// TIA Portal V19 program export: 1 tag tables, 1 data types, 2 data blocks, 10 code blocks (in call order from the OBs), 4 instance data blocks

VAR_GLOBAL   // PLC tag table "DefaultTagTable"
   Tag_1 AT %M20.7 : Bool;
END_VAR

TYPE "typeStartLift"
TITLE = typeStartLift
// PLC data type start lift
   STRUCT
      startLiftUp : Bool;   // Start lift up
      startLiftDown : Bool;   // Start lift down
   END_STRUCT;
END_TYPE

DATA_BLOCK "Actions"   // DB3
{ S7_Optimized_Access := 'TRUE' }
// stored: MemoryReserve 100
   VAR
      Action_AirComprID1 : String := 'Check that no emergency stop has been depressed. If it has, check why. The machine is now ready to start with the Unit On button. The alarm is reset automatically when the cause is removed (logically controlled).';
      TextList : DWord;
      Trigger : UInt;
      Ack : Bool;
   END_VAR
BEGIN
END_DATA_BLOCK

DATA_BLOCK "SeqData"   // DB11
TITLE = SeqData
{ S7_Optimized_Access := 'TRUE'; DB_Accessible_From_OPC_UA := 'FALSE' }
AUTHOR : Siemens
// Global DB for BeltLift
// stored: DBAccessibleFromOPCUA false, MemoryReserve 100
   VAR
      plantOn : Bool := true;   // Plant switched on
      compressedAir : Bool;   // Druckluft nicht in Ordnung. Im Fehlerfall ist die Ursache: Der zur Maschine gehörende Not-Halt hat die Maschine gestoppt. Bei ausgeschalteter Maschine oder gedrücktem Not-Halt können keine Funktionen ausgeführt werden. / Compressed air not OK. In case of an Error Cause: The emergency stop belonging to the machine has stopped the machine. No functions can be performed when the machine is shut off or the emergency stop is pressed.
      powerVoltage : Bool;   // Spannungsversorgung nicht in Ordnung. Im Fehlerfall ist die Druckluft nicht in Ordnung. Im Fehlerfall ist die Ursache: Der zur Maschine gehörende Not-Halt hat die Maschine gestoppt. Bei ausgeschalteter Maschine oder gedrücktem Not-Halt können keine Funktionen ausgeführt werden. / Voltage power supply not OK.
      doorClosed : Bool;   // Safety door closed
      autoStart : Bool;   // Automatic start
      autoStop : Bool;   // Automatic stop
      autoStarted : Bool := false;   // Automatic started
      autoStopped : Bool;   // Automatic stopped
      ackSeq : Bool;   // Acknowledge GRAPH FB
      errFltSeq : Bool;   // Error Graph FB
      seqStart : Bool;   // GRAPH sequence started
      newCase : Bool;   // Sensor new case
      posCaseBelt : Int;   // Case position on belt
      posLift1 : Int;   // Lift 1 position
      posLift2 : Int;   // Lift 2 position
      visCaseLift1 : Bool;   // Case lift1 visible
      visCaseLift2 : Bool;   // Case lift2 visible
      setStop1 : Bool;   // Set stopper1
      setStop2 : Bool;   // Set stopper2
      sensorStop1 : Bool;   // Sensor at stopper1
      sensorStop2 : Bool;   // Sensor at stopper2
      sensorStop3 : Bool;   // Sensor at stopper3
      errSensorStop1 : Bool;   // Error on Sensor at stopper1
      errSensorStop2 : Bool;   // Error on Sensor at stopper2
      errSensorStop3 : Bool;   // Error on Sensor at stopper2
      errSensorNewCase : Bool;   // Error on Sensor at new case
      toLift1 : Bool;   // Case to lift1 or lift2
      autoLift1 : "typeStartLift";   // Start automatic lift1
      autoLift2 : "typeStartLift";   // Start automatic lift2
      manLift1 : "typeStartLift";   // Start manual lift1
      manLift2 : "typeStartLift";   // Start manual lift2
      outLift1Up : Bool;   // Output lift1 up
      outLift1Down : Bool;   // Output lift1 down
      outLift2Up : Bool;   // Output lift2 up
      outLift2Down : Bool;   // Output lift2 down
      sensorLift1Up : Bool;   // Sensor lift1 up
      sensorLift1Down : Bool;   // Sensor lift1 down
      sensorLift2Up : Bool;   // Sensor lift2 up
      sensorLift2Down : Bool;   // Sensor lift2 down
      simOperandSupVis : Bool;   // Simulation supervision operand
      simInterlockSupVis : Bool;   // Simulation supervision interlock
      simLiftFreeSupVis : Bool;   // Simulation supervision lift free
      simActReactSupVis : Bool;   // Simulation supervision action and reaction
      simPositionSupVis : Bool;   // Simulation supervision position
      simUdtOperandSupVis : Bool;   // Simulation supervision operand in UDT
      simActive : Bool;   // Simulation active
      releaseSimPlantOn : Bool;   // Release simulation plant on
      releaseSimAutoStarted : Bool;   // Release simulation auto started
      releaseSimAutoStopped : Bool;   // Release simulation auto stopped
      beltLEDs : Word;   // Moving lights belt
      lift1LEDs : Word;   // Moving lights lift1
      lift2LEDs : Word;   // Moving lights lift2
      stateCase : Array[0..3] of Bool;   // State case position
      liftFree : Bool := true;   // Lift is free for new case / Lift ist bereit für einen neuen Kasten
      simInterlockSupVisLiftFree : Bool;   // Simulation supervision interlock / Simulation supervision interlock lift free
      resetCrit : Bool;
      identTimeStamp : LDT;
      retVal : Int;
      frequency : Real := 10.0;
      freqError : Bool;
      freqStatus : Word;
      textListID { ExternalAccessible := 'False'; ExternalVisible := 'False'; ExternalWritable := 'False'} : Word;
   END_VAR
BEGIN
END_DATA_BLOCK

ORGANIZATION_BLOCK "Main"   // OB1, LAD, ProgramCycle
TITLE = "Main Program Sweep (Cycle)"
{ S7_Optimized_Access := 'TRUE' }
AUTHOR : Siemens
// "Main Program
// stored: IsIECCheckEnabled true, SetENOAutomatically true
   VAR_INPUT
      Initial_Call : Bool;   // Initial call of this OB
      Remanence : Bool;   // =True, if remanent data are available
   END_VAR
BEGIN

REGION Network 1
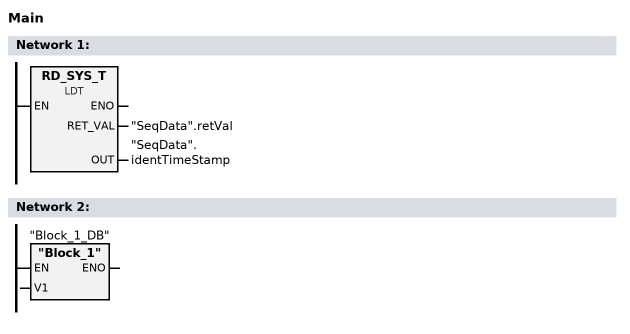
   RUNG wire#powerrail
      { S7_Templates := "date_type := LDT" } RD_SYS_T(RET_VAL => "SeqData".retVal, OUT => "SeqData".identTimeStamp)
   END_RUNG
   // the same network as SCL:
   "SeqData".retVal := RD_SYS_T(OUT => "SeqData".identTimeStamp);
END_REGION

REGION Network 2
   RUNG wire#powerrail
      "Block_1_DB"(V1 :=)
   END_RUNG
   // the same network as SCL:
   "Block_1_DB"();   // "Block_1"
END_REGION
END_ORGANIZATION_BLOCK

ORGANIZATION_BLOCK "MainBeltLift"   // OB125, FBD, ProgramCycle
TITLE = "Main Program Sweep (Cycle)"
{ S7_Optimized_Access := 'TRUE' }
AUTHOR : Siemens
// Main programm belt lift
// stored: IsIECCheckEnabled true, SetENOAutomatically true
   VAR_INPUT
      Initial_Call : Bool;   // Initial call of this OB
      Remanence : Bool;   // =True, if remanent data are available
   END_VAR
BEGIN

REGION Network 1
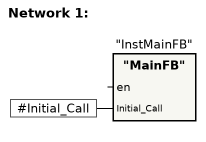
   "InstMainFB"(Initial_Call := #Initial_Call);   // "MainFB"
END_REGION
END_ORGANIZATION_BLOCK

FUNCTION_BLOCK "MainFB"   // FB10, FBD
TITLE = MainFB
{ S7_Optimized_Access := 'TRUE' }
AUTHOR : Siemens
// Main FB BeltLift
// stored: IsIECCheckEnabled true, MemoryReserve 100, SetENOAutomatically true
   VAR_INPUT
      Initial_Call { ExternalAccessible := 'False'; ExternalVisible := 'False'; ExternalWritable := 'False'} : Bool;   // Initial call of this OB
   END_VAR
   VAR
      instCommon { ExternalAccessible := 'False'; ExternalVisible := 'False'; ExternalWritable := 'False'; S7_SetPoint := 'True'} : "Common";
      instLift1Cmd { ExternalAccessible := 'False'; ExternalVisible := 'False'; ExternalWritable := 'False'; S7_SetPoint := 'True'} : "LiftCmd";
      instLift2Cmd { ExternalAccessible := 'False'; ExternalVisible := 'False'; ExternalWritable := 'False'; S7_SetPoint := 'True'} : "LiftCmd";
      instLiftSim { ExternalAccessible := 'False'; ExternalVisible := 'False'; ExternalWritable := 'False'; S7_SetPoint := 'True'} : "LiftSim";
   END_VAR
BEGIN

REGION Network 1: common
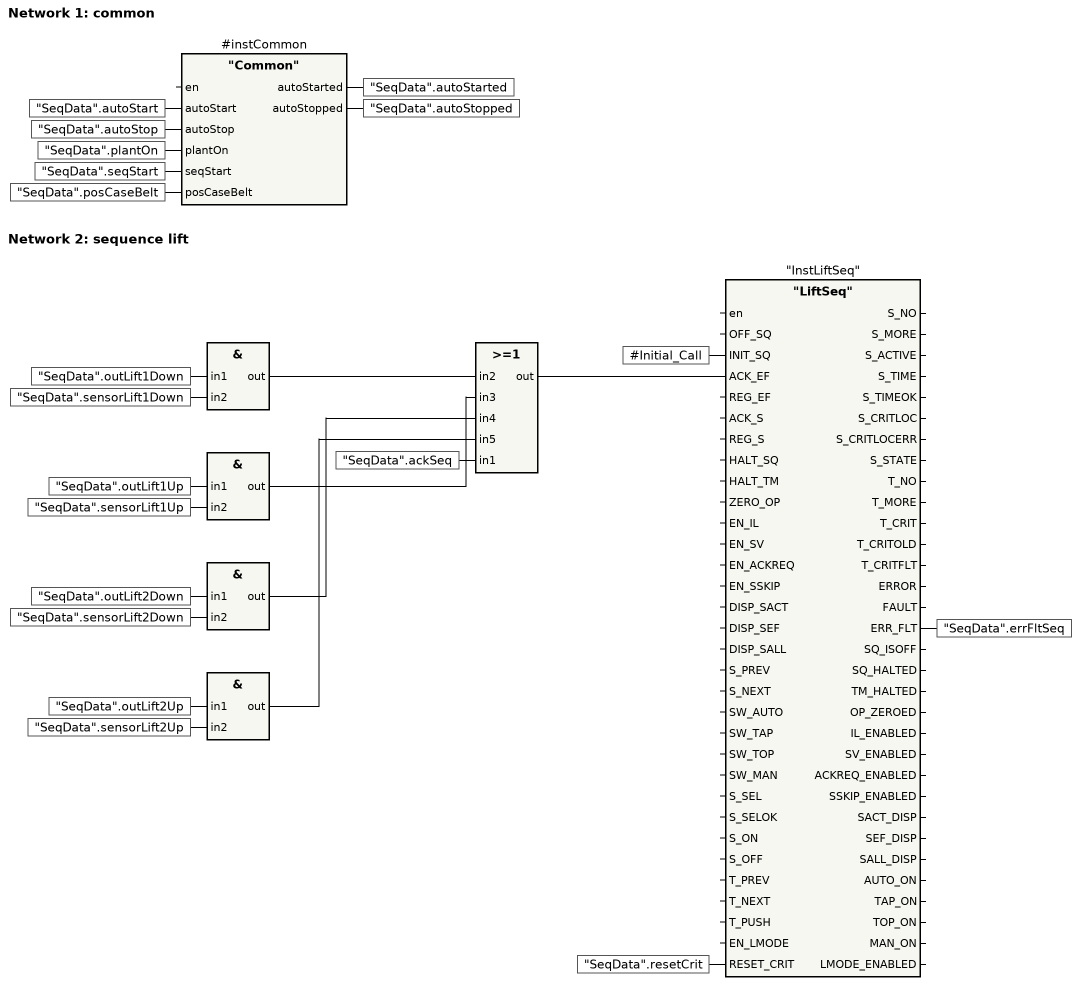
   #instCommon(autoStart := "SeqData".autoStart,   // "Common"
               autoStop := "SeqData".autoStop,
               plantOn := "SeqData".plantOn,
               seqStart := "SeqData".seqStart,
               posCaseBelt := "SeqData".posCaseBelt,
               autoStarted => "SeqData".autoStarted,
               autoStopped => "SeqData".autoStopped);
END_REGION

REGION Network 2: sequence lift
   "InstLiftSeq"(INIT_SQ := #Initial_Call,   // "LiftSeq"
                 ACK_EF := ("SeqData".outLift1Down AND "SeqData".sensorLift1Down) OR ("SeqData".outLift1Up AND "SeqData".sensorLift1Up) OR ("SeqData".outLift2Down AND "SeqData".sensorLift2Down) OR ("SeqData".outLift2Up AND "SeqData".sensorLift2Up) OR "SeqData".ackSeq,
                 RESET_CRIT := "SeqData".resetCrit,
                 ERR_FLT => "SeqData".errFltSeq);
END_REGION

REGION Network 3: Lift 1
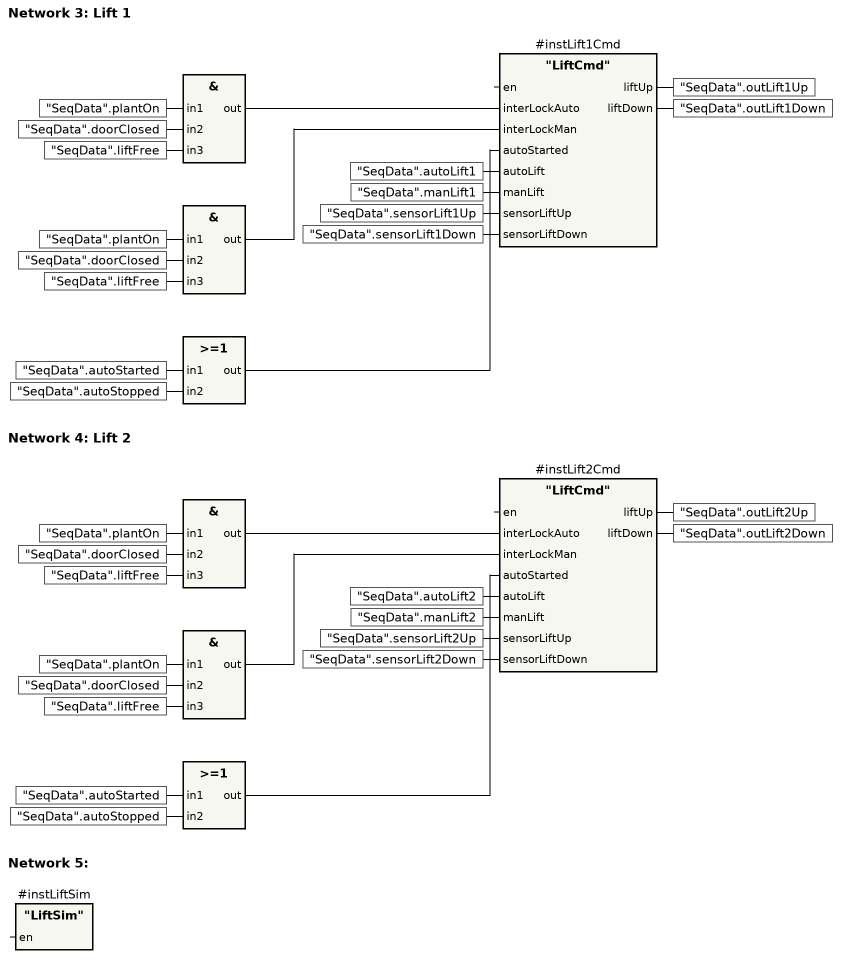
   #instLift1Cmd(interLockAuto := "SeqData".plantOn AND "SeqData".doorClosed AND "SeqData".liftFree,   // "LiftCmd"
                 interLockMan := "SeqData".plantOn AND "SeqData".doorClosed AND "SeqData".liftFree,
                 autoStarted := "SeqData".autoStarted OR "SeqData".autoStopped,
                 autoLift := "SeqData".autoLift1,
                 manLift := "SeqData".manLift1,
                 sensorLiftUp := "SeqData".sensorLift1Up,
                 sensorLiftDown := "SeqData".sensorLift1Down,
                 liftUp => "SeqData".outLift1Up,
                 liftDown => "SeqData".outLift1Down);
END_REGION

REGION Network 4: Lift 2
   #instLift2Cmd(interLockAuto := "SeqData".plantOn AND "SeqData".doorClosed AND "SeqData".liftFree,   // "LiftCmd"
                 interLockMan := "SeqData".plantOn AND "SeqData".doorClosed AND "SeqData".liftFree,
                 autoStarted := "SeqData".autoStarted OR "SeqData".autoStopped,
                 autoLift := "SeqData".autoLift2,
                 manLift := "SeqData".manLift2,
                 sensorLiftUp := "SeqData".sensorLift2Up,
                 sensorLiftDown := "SeqData".sensorLift2Down,
                 liftUp => "SeqData".outLift2Up,
                 liftDown => "SeqData".outLift2Down);
END_REGION

REGION Network 5
   #instLiftSim();   // "LiftSim"
END_REGION
END_FUNCTION_BLOCK

FUNCTION_BLOCK "Common"   // FB13, FBD
TITLE = Common
{ S7_Optimized_Access := 'TRUE' }
AUTHOR : Siemens
// Common functions BeltLift
// stored: IsIECCheckEnabled true, MemoryReserve 100, SetENOAutomatically true
   VAR_INPUT
      autoStart { ExternalAccessible := 'False'; ExternalVisible := 'False'; ExternalWritable := 'False'} : Bool;
      autoStop { ExternalAccessible := 'False'; ExternalVisible := 'False'; ExternalWritable := 'False'} : Bool;
      plantOn { ExternalAccessible := 'False'; ExternalVisible := 'False'; ExternalWritable := 'False'} : Bool;
      seqStart { ExternalAccessible := 'False'; ExternalVisible := 'False'; ExternalWritable := 'False'} : Bool;
      posCaseBelt { ExternalAccessible := 'False'; ExternalVisible := 'False'; ExternalWritable := 'False'} : Int;
   END_VAR
   VAR_OUTPUT
      autoStarted { ExternalAccessible := 'False'; ExternalVisible := 'False'; ExternalWritable := 'False'} : Bool;
      autoStopped { ExternalAccessible := 'False'; ExternalVisible := 'False'; ExternalWritable := 'False'} : Bool;
   END_VAR
   VAR
      statCaseOnStopper { ExternalAccessible := 'False'; ExternalVisible := 'False'; ExternalWritable := 'False'} : Bool;
      statAutoStopped { ExternalAccessible := 'False'; ExternalVisible := 'False'; ExternalWritable := 'False'} : Bool;
   END_VAR
BEGIN

REGION Network 1
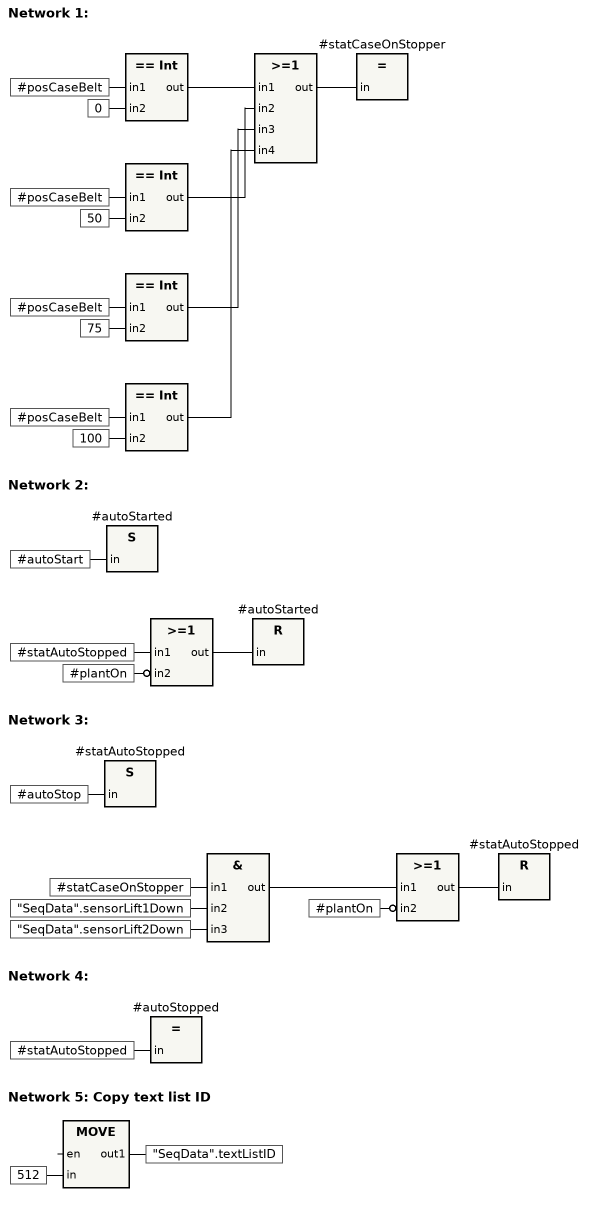
   #statCaseOnStopper := (#posCaseBelt = 0) OR (#posCaseBelt = 50) OR (#posCaseBelt = 75) OR (#posCaseBelt = 100);
END_REGION

REGION Network 2
   IF #autoStart THEN #autoStarted := TRUE; END_IF;
   IF #statAutoStopped OR NOT #plantOn THEN #autoStarted := FALSE; END_IF;
END_REGION

REGION Network 3
   IF #autoStop THEN #statAutoStopped := TRUE; END_IF;
   IF (#statCaseOnStopper AND "SeqData".sensorLift1Down AND "SeqData".sensorLift2Down) OR NOT #plantOn THEN
       #statAutoStopped := FALSE;
   END_IF;
END_REGION

REGION Network 4
   #autoStopped := #statAutoStopped;
END_REGION

REGION Network 5: Copy text list ID
   "SeqData".textListID := 512;
END_REGION
END_FUNCTION_BLOCK

FUNCTION_BLOCK "LiftSeq"   // FB12, GRAPH
TITLE = LiftSeq
AUTHOR : Siemens
// Graph sequence BeltLift
// stored: GraphVersion 6.0, InitialValuesAcquisition true, IsIECCheckEnabled true, LanguageInNetworks FBD, SetENOAutomatically true
   // inherited from GRAPH_BASE
   VAR_INPUT
      OFF_SQ { ExternalWritable := 'False'} : Bool := false;   // Kette ausschalten / Turn sequence off
      INIT_SQ { ExternalWritable := 'False'} : Bool := false;   // Kette in Initialzustand versetzen / Set sequence to initial state
      ACK_EF { ExternalWritable := 'False'} : Bool := false;   // Alle Fehler und Störungen quittieren / Acknowledge all errors and faults
      REG_EF { ExternalWritable := 'False'} : Bool := false;   // Register all errors and faults / Alle Fehler und Störungen registrieren
      ACK_S { ExternalWritable := 'False'} : Bool := false;   // Acknowledge step indicated in S_NO / Schritt quittieren, der an Parameter S_NO anliegt
      REG_S { ExternalWritable := 'False'} : Bool := false;   // Register the step indicated in S_NO / Schritt registrieren, der an Parameter S_NO anliegt
      HALT_SQ { ExternalWritable := 'False'} : Bool := false;   // Halt sequence immediately / Kette sofort anhalten
      HALT_TM { ExternalWritable := 'False'} : Bool := false;   // Halt timers immediately / Zeiten sofort anhalten
      ZERO_OP { ExternalWritable := 'False'} : Bool := false;   // Set all operands assigned with N, L, D to 0 / Alle mit N, L, D zugewiesenen Operanden auf 0 setzen
      EN_IL { ExternalWritable := 'False'} : Bool := false;   // Activate interlocks / Interlockbearbeitung aktivieren
      EN_SV { ExternalWritable := 'False'} : Bool := false;   // Activate supervision processing / Supervisionsbearbeitung aktivieren
      EN_ACKREQ { ExternalWritable := 'False'} : Bool := false;   // Activate mandatory acknowledgment / Quittierpflicht aktivieren
      EN_SSKIP { ExternalWritable := 'False'} : Bool := false;   // Enable "Skip step" / "Schritte überspringen" aktivieren
      DISP_SACT { ExternalWritable := 'False'} : Bool := false;   // Display active steps only / Nur aktive Schritte anzeigen
      DISP_SEF { ExternalWritable := 'False'} : Bool := false;   // Display only steps with errors and disrupted steps / Nur fehlerhafte und gestörte Schritte anzeigen
      DISP_SALL { ExternalWritable := 'False'} : Bool := false;   // Display all steps / Alle Schritte anzeigen
      S_PREV { ExternalWritable := 'False'} : Bool := false;   // Vorherigen Schritt am Parameter S_NO ausgeben / Output previous step in parameter S_NO
      S_NEXT { ExternalWritable := 'False'} : Bool := false;   // Nächsten Schritt am Parameter S_NO anzeigen / Indicate next step in parameter S_NO
      SW_AUTO { ExternalWritable := 'False'} : Bool := false;   // Automtischer Betrieb / Automatic mode
      SW_TAP { ExternalWritable := 'False'} : Bool := false;   // Halbautomatisch/Weiterschalten mit Transition / Semiautomatic/switch with transition
      SW_TOP { ExternalWritable := 'False'} : Bool := false;   // Halbautomatisch/Ignoriere Transition / Semiautomatic/ignore transition
      SW_MAN { ExternalWritable := 'False'} : Bool := false;   // Handbetrieb / Manual mode
      S_SEL { ExternalWritable := 'False'} : Int := 0;   // Schritt auswählen, der an S_NO ausgegeben werden soll / Select step to be output to S_NO
      S_SELOK { ExternalWritable := 'False'} : Bool := false;   // Enter value from S_SEL in S_NO / Wert aus S_SEL nach S_NO übernehmen
      S_ON { ExternalWritable := 'False'} : Bool := false;   // Schritt aktivieren, der an Parameter S_NO anliegt / Activate step indicated in S_NO
      S_OFF { ExternalWritable := 'False'} : Bool := false;   // Schritt deaktivieren, der an Parameter S_NO anliegt / Deactivate step indicated S_NO
      T_PREV { ExternalWritable := 'False'} : Bool := false;   // Display previous transition in T_NO / Vorherige Transition an Parameter T_NO anzeigen
      T_NEXT { ExternalWritable := 'False'} : Bool := false;   // Display next transition at parameter T_NO / Nächste Transition an Parameter T_NO anzeigen
      T_PUSH { ExternalWritable := 'False'} : Bool := false;   // Schaltfreigabe für Transition im halbautomatischen Betrieb / Enable transition to switch in semi automatic mode
      EN_LMODE { ExternalWritable := 'False'} : Bool := false;   // Activate learning mode / Lernmodus aktivieren
      RESET_CRIT { ExternalWritable := 'False'} : Bool := false;   // Reset all initial values recorded for interlocks and transitions / Alle Erstwerte, die für Interlocks und Transitionen aufgezeichnet wurden, zurücksetzen
   END_VAR
   VAR_OUTPUT
      S_NO { ExternalWritable := 'False'} : Int := 0;   // Schrittnummer / Step number
      S_MORE { ExternalWritable := 'False'} : Bool := false;   // Weitere Schritte sind vorhanden und können in S_NO angezeigt werden. / More steps are available and can be shown in S_NO
      S_ACTIVE { ExternalWritable := 'False'} : Bool := false;   // Schritt, der an Parameter S_NO angezeigt wird, ist aktiv / Step indicated in S_NO is active
      S_TIME { ExternalWritable := 'False'} : Time := T#0ms;   // Step activation time / Schrittaktivierungszeit
      S_TIMEOK { ExternalWritable := 'False'} : Time := T#0ms;   // No error in step activation time / Schrittaktivierungszeit fehlerfrei
      S_CRITLOC { ExternalWritable := 'False'} : DWord := 16#0;   // Interlock criteria bits / Interlock-Kriterienbits
      S_CRITLOCERR { ExternalWritable := 'False'} : DWord := 16#0;   // Interlock criteria bits for event L1 / Interlock-Kriterienbits bei Ereignis L1
      S_STATE { ExternalWritable := 'False'} : Word := 16#0;   // Step state bits / Schrittzustandsbits
      T_NO { ExternalWritable := 'False'} : Int := 0;   // Transition number / Transitionsnummer
      T_MORE { ExternalWritable := 'False'} : Bool := false;   // More valid transitions available for display / Weitere gültige Transitionen zur Anzeige verfügbar
      T_CRIT { ExternalWritable := 'False'} : DWord := 16#0;   // Transition criteria bits / Transitions-Kriterienbits
      T_CRITOLD { ExternalWritable := 'False'} : DWord := 16#0;   // Transition criteria bits from last cycle / Transitions-Kriterienbits des letzten Zyklus
      T_CRITFLT { ExternalWritable := 'False'} : DWord := 16#0;   // Transition criteria bits for event V1 / Transitions-Kriterienbits bei Ereignis V1
      ERROR { ExternalWritable := 'False'} : Bool := false;   // Interlock group error / Sammelfehler Interlock
      FAULT { ExternalWritable := 'False'} : Bool := false;   // Supervision group error / Sammelfehler Supervision
      ERR_FLT { ExternalWritable := 'False'} : Bool := false;   // Sammelfehler Interlock oder Supervision / Interlock or supervision group error
      SQ_ISOFF { ExternalWritable := 'False'} : Bool := false;   // Sequence is off (no step active) / Kette ausgeschaltet (kein Schritt aktiv)
      SQ_HALTED { ExternalWritable := 'False'} : Bool := false;   // Sequence halted / Kette angehalten
      TM_HALTED { ExternalWritable := 'False'} : Bool := false;   // Timers halted / Zeiten angehalten
      OP_ZEROED { ExternalWritable := 'False'} : Bool := false;   // All the operands assigned with N, L, D are set to 0 / Alle mit N, L oder D zugewiesenen Operanden auf 0 gesetzt
      IL_ENABLED { ExternalWritable := 'False'} : Bool := false;   // Interlocks are active / Interlockbearbeitung aktiv
      SV_ENABLED { ExternalWritable := 'False'} : Bool := false;   // Supervision processing activated / Supervisionsbearbeitung aktiviert
      ACKREQ_ENABLED { ExternalWritable := 'False'} : Bool := false;   // Mandatory acknowledgment activated / Quittierpflicht aktiviert
      SSKIP_ENABLED { ExternalWritable := 'False'} : Bool := false;   // Skip steps activated / Schritte überspringen aktiviert
      SACT_DISP { ExternalWritable := 'False'} : Bool := false;   // Display active steps only / Nur aktive Schritte anzeigen
      SEF_DISP { ExternalWritable := 'False'} : Bool := false;   // Display only steps with errors or disrupted steps / Nur fehlerhafte oder gestörte Schritte anzeigen
      SALL_DISP { ExternalWritable := 'False'} : Bool := false;   // Display all steps / Alle Schritte anzeigen
      AUTO_ON { ExternalWritable := 'False'} : Bool := false;   // Automatischer Betrieb eingeschaltet / Automatic mode is active
      TAP_ON { ExternalWritable := 'False'} : Bool := false;   // Halbautomatischer Betrieb/Schritt mit Transition eingeschaltet / Semiautomatic mode/step with transition enabled
      TOP_ON { ExternalWritable := 'False'} : Bool := false;   // Halbautomatischer Betrieb/Ignoriere Transition eingeschaltet / Semiautomatic mode/ignore transition enabled
      MAN_ON { ExternalWritable := 'False'} : Bool := false;   // Handbetrieb eingeschaltet / Manual mode is active
      LMODE_ENABLED { ExternalWritable := 'False'} : Bool := false;   // Learning mode is active / Lernmodus aktiv
   END_VAR
BEGIN
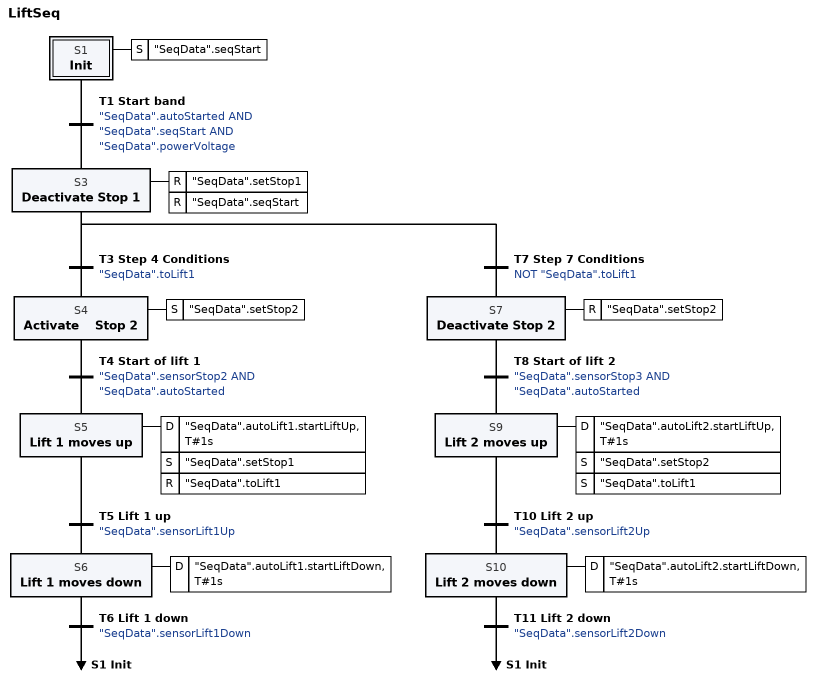
   // sequencer 1
   INITIAL_STEP Init:   // S1, max time T#10S, warning time T#7S
              S    "SeqData".seqStart
   END_STEP
   TRANSITION "Start band" FROM Init TO "Deactivate Stop 1"   // T1
      := "SeqData".autoStarted AND "SeqData".seqStart AND "SeqData".powerVoltage;
   END_TRANSITION
   STEP "Deactivate Stop 1":   // S3, max time T#10S, warning time T#7S
              R    "SeqData".setStop1
              R    "SeqData".seqStart
   END_STEP
   TRANSITION "Step 4 Conditions" FROM "Deactivate Stop 1" TO "Activate    Stop 2"   // T3
      := "SeqData".toLift1;
   END_TRANSITION
   TRANSITION "Step 7 Conditions" FROM "Deactivate Stop 1" TO "Deactivate Stop 2"   // T7
      := NOT "SeqData".toLift1;
   END_TRANSITION
   STEP "Activate    Stop 2":   // S4, max time T#10S, warning time T#7S
              S    "SeqData".setStop2
   END_STEP
   TRANSITION "Start of lift 1" FROM "Activate    Stop 2" TO "Lift 1 moves up"   // T4
      := "SeqData".sensorStop2 AND "SeqData".autoStarted;
   END_TRANSITION
   STEP "Lift 1 moves up":   // S5, max time T#10S, warning time T#7S
      interlock C := "SeqData".doorClosed AND "SeqData".liftFree;   // Door at lift not closed or lift blocked. / Tür an Hubeinheit nicht geschlossen oder Hubeinheit blockiert.
      supervision V := #"Lift 1 moves up".T > T#5S;   // Lift1 upper position not reached / Hubeinheit 1obere Position nicht erreicht
              D    "SeqData".autoLift1.startLiftUp, T#1s
              S    "SeqData".setStop1
              R    "SeqData".toLift1
   END_STEP
   TRANSITION "Lift 1 up" FROM "Lift 1 moves up" TO "Lift 1 moves down"   // T5
      := "SeqData".sensorLift1Up;
   END_TRANSITION
   STEP "Lift 1 moves down":   // S6, max time T#10S, warning time T#7S
      interlock C := "SeqData".doorClosed AND "SeqData".liftFree;   // Door at lift not closed or lift blocked. / Tür an Hubeinheit nicht geschlossen oder Hubeinheit blockiert.
      supervision V := #"Lift 1 moves down".T > T#5S;   // Lift1 lower position not reached / Hubeinheit 1 untere Position nicht erreicht
              D    "SeqData".autoLift1.startLiftDown, T#1s
   END_STEP
   TRANSITION "Lift 1 down" FROM "Lift 1 moves down" TO Init   // T6, jump
      := "SeqData".sensorLift1Down;
   END_TRANSITION
   STEP "Deactivate Stop 2":   // S7, max time T#10S, warning time T#7S
              R    "SeqData".setStop2
   END_STEP
   TRANSITION "Start of lift 2" FROM "Deactivate Stop 2" TO "Lift 2 moves up"   // T8
      := "SeqData".sensorStop3 AND "SeqData".autoStarted;
   END_TRANSITION
   STEP "Lift 2 moves up":   // S9, max time T#10S, warning time T#7S
      interlock C := "SeqData".doorClosed AND "SeqData".liftFree;   // Door at lift not closed or lift blocked. / Tür an Hubeinheit nicht geschlossen oder Hubeinheit blockiert.
      supervision V := #"Lift 2 moves up".T > T#5S;   // Lift2 upper position not reached / Hubeinheit 2 obere Position nicht erreicht
              D    "SeqData".autoLift2.startLiftUp, T#1s
              S    "SeqData".setStop2
              S    "SeqData".toLift1
   END_STEP
   TRANSITION "Lift 2 up" FROM "Lift 2 moves up" TO "Lift 2 moves down"   // T10
      := "SeqData".sensorLift2Up;
   END_TRANSITION
   STEP "Lift 2 moves down":   // S10, max time T#10S, warning time T#7S
      interlock C := "SeqData".doorClosed AND "SeqData".liftFree;   // Door at lift not closed or lift blocked. / Tür an Hubeinheit nicht geschlossen oder Hubeinheit blockiert.
      supervision V := #"Lift 2 moves down".T > T#5S;   // Lift2 lower position not reached / Hubeinheit 2 untere Position nicht erreicht
              D    "SeqData".autoLift2.startLiftDown, T#1s
   END_STEP
   TRANSITION "Lift 2 down" FROM "Lift 2 moves down" TO Init   // T11, jump
      := "SeqData".sensorLift2Down;
   END_TRANSITION
END_FUNCTION_BLOCK

FUNCTION_BLOCK "LiftCmd"   // FB11, LAD
TITLE = LiftCmd
{ S7_Optimized_Access := 'TRUE' }
AUTHOR : Siemens
// Lift command BeltLift
// stored: IsIECCheckEnabled true, MemoryReserve 100, SetENOAutomatically true
   VAR_INPUT
      interLockAuto { ExternalAccessible := 'False'; ExternalVisible := 'False'; ExternalWritable := 'False'} : Bool;   // Interlock automatic
      interLockMan { ExternalAccessible := 'False'; ExternalVisible := 'False'; ExternalWritable := 'False'} : Bool;   // Interlock manual
      autoStarted { ExternalAccessible := 'False'; ExternalVisible := 'False'; ExternalWritable := 'False'} : Bool;   // Automatic started
      autoLift { ExternalAccessible := 'False'; ExternalVisible := 'False'; ExternalWritable := 'False'} : "typeStartLift";   // Start auto lift
      manLift { ExternalAccessible := 'False'; ExternalVisible := 'False'; ExternalWritable := 'False'} : "typeStartLift";   // Start manual lift
      sensorLiftUp { ExternalAccessible := 'False'; ExternalVisible := 'False'; ExternalWritable := 'False'} : Bool;   // Sensor lift up
      sensorLiftDown { ExternalAccessible := 'False'; ExternalVisible := 'False'; ExternalWritable := 'False'} : Bool;   // Sensor lift down
   END_VAR
   VAR_OUTPUT
      liftUp { ExternalAccessible := 'False'; ExternalVisible := 'False'; ExternalWritable := 'False'} : Bool;   // Output lift up
      liftDown { ExternalAccessible := 'False'; ExternalVisible := 'False'; ExternalWritable := 'False'} : Bool;   // Output lift down
   END_VAR
   VAR
      statTrigLift { ExternalAccessible := 'False'; ExternalVisible := 'False'; ExternalWritable := 'False'} : "typeStartLift";   // Trigger lift up / Trigger lift
   END_VAR
BEGIN

REGION Network 1: set trigger lift up
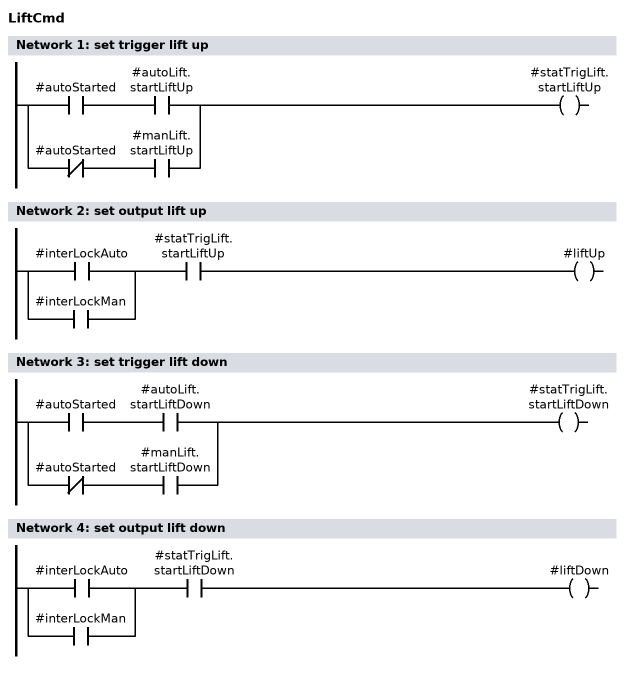
   RUNG wire#powerrail
      Contact( #autoStarted )
      Contact( #autoLift.startLiftUp )
      wire#w1
      Coil( #statTrigLift.startLiftUp )
   END_RUNG
   RUNG wire#powerrail
      I_Contact( #autoStarted )
      Contact( #manLift.startLiftUp )
   END_RUNG wire#w1
   // the same network as SCL:
   #statTrigLift.startLiftUp := (#autoStarted AND #autoLift.startLiftUp) OR (NOT #autoStarted AND #manLift.startLiftUp);
END_REGION

REGION Network 2: set output lift up
   RUNG wire#powerrail
      Contact( #interLockAuto )
      wire#w1
      Contact( #statTrigLift.startLiftUp )
      Coil( #liftUp )
   END_RUNG
   RUNG wire#powerrail
      Contact( #interLockMan )
   END_RUNG wire#w1
   // the same network as SCL:
   #liftUp := (#interLockAuto OR #interLockMan) AND #statTrigLift.startLiftUp;
END_REGION

REGION Network 3: set trigger lift down
   RUNG wire#powerrail
      Contact( #autoStarted )
      Contact( #autoLift.startLiftDown )
      wire#w1
      Coil( #statTrigLift.startLiftDown )
   END_RUNG
   RUNG wire#powerrail
      I_Contact( #autoStarted )
      Contact( #manLift.startLiftDown )
   END_RUNG wire#w1
   // the same network as SCL:
   #statTrigLift.startLiftDown := (#autoStarted AND #autoLift.startLiftDown) OR (NOT #autoStarted AND #manLift.startLiftDown);
END_REGION

REGION Network 4: set output lift down
   RUNG wire#powerrail
      Contact( #interLockAuto )
      wire#w1
      Contact( #statTrigLift.startLiftDown )
      Coil( #liftDown )
   END_RUNG
   RUNG wire#powerrail
      Contact( #interLockMan )
   END_RUNG wire#w1
   // the same network as SCL:
   #liftDown := (#interLockAuto OR #interLockMan) AND #statTrigLift.startLiftDown;
END_REGION
END_FUNCTION_BLOCK

FUNCTION_BLOCK "LiftSim"   // FB14, FBD
TITLE = LiftSim
{ S7_Optimized_Access := 'TRUE' }
AUTHOR : Siemens
// Simulation BeltLift
// stored: IsIECCheckEnabled true, MemoryReserve 100, SetENOAutomatically true
   VAR
      instRisTrigLift1 { ExternalAccessible := 'False'; ExternalVisible := 'False'; ExternalWritable := 'False'; S7_SetPoint := 'True'} : R_TRIG;
      instRisTrigLift2 { ExternalAccessible := 'False'; ExternalVisible := 'False'; ExternalWritable := 'False'; S7_SetPoint := 'True'} : R_TRIG;
      statRisTrigLift1 { ExternalAccessible := 'False'; ExternalVisible := 'False'; ExternalWritable := 'False'} : Bool;
      statRisTrigLift2 { ExternalAccessible := 'False'; ExternalVisible := 'False'; ExternalWritable := 'False'} : Bool;
      instRisTrigClock { ExternalAccessible := 'False'; ExternalVisible := 'False'; ExternalWritable := 'False'; S7_SetPoint := 'True'} : R_TRIG;
      statRisTrigClock { ExternalAccessible := 'False'; ExternalVisible := 'False'; ExternalWritable := 'False'} : Bool;
      statClock10Hz { ExternalAccessible := 'False'; ExternalVisible := 'False'; ExternalWritable := 'False'} : Bool;
      instMovingLightBelt { ExternalAccessible := 'False'; ExternalVisible := 'False'; ExternalWritable := 'False'; S7_SetPoint := 'True'} : "MovingLight";
      instMovingLightLift1 { ExternalAccessible := 'False'; ExternalVisible := 'False'; ExternalWritable := 'False'; S7_SetPoint := 'True'} : "MovingLight";
      instMovingLightLift2 { ExternalAccessible := 'False'; ExternalVisible := 'False'; ExternalWritable := 'False'; S7_SetPoint := 'True'} : "MovingLight";
      statDirBelt { ExternalAccessible := 'False'; ExternalVisible := 'False'; ExternalWritable := 'False'} : Int;
      statDirLift1 { ExternalAccessible := 'False'; ExternalVisible := 'False'; ExternalWritable := 'False'} : Int;
      statDirLift2 { ExternalAccessible := 'False'; ExternalVisible := 'False'; ExternalWritable := 'False'} : Int;
      instLEDsBelt { ExternalAccessible := 'False'; ExternalVisible := 'False'; ExternalWritable := 'False'; S7_SetPoint := 'True'} : "LEDs";
      instLEDsLift1 { ExternalAccessible := 'False'; ExternalVisible := 'False'; ExternalWritable := 'False'; S7_SetPoint := 'True'} : "LEDs";
      instLEDsLift2 { ExternalAccessible := 'False'; ExternalVisible := 'False'; ExternalWritable := 'False'; S7_SetPoint := 'True'} : "LEDs";
   END_VAR
BEGIN

REGION Network 1
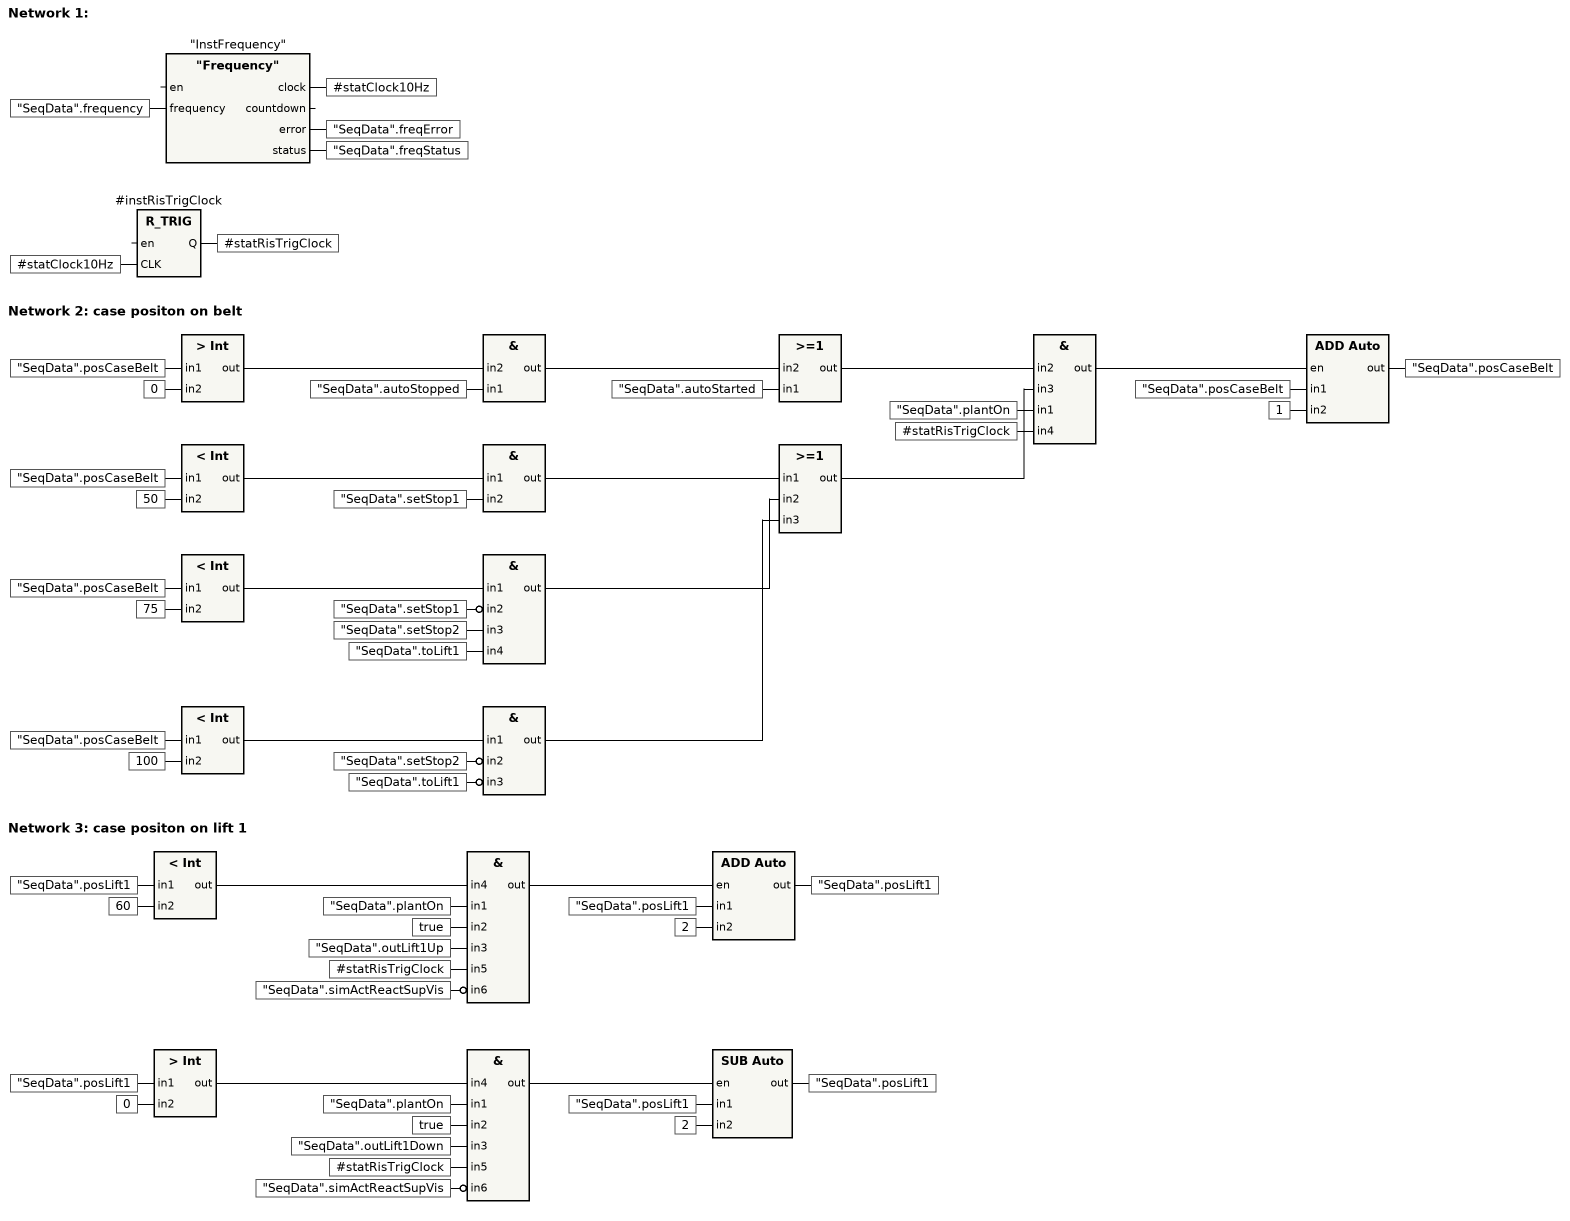
   "InstFrequency"(frequency := "SeqData".frequency,   // "Frequency"
                   clock => #statClock10Hz,
                   error => "SeqData".freqError,
                   status => "SeqData".freqStatus);
   #instRisTrigClock(CLK := #statClock10Hz, Q => #statRisTrigClock);   // R_TRIG
END_REGION

REGION Network 2: case positon on belt
   IF ((("SeqData".posCaseBelt > 0) AND "SeqData".autoStopped) OR "SeqData".autoStarted) AND ((("SeqData".posCaseBelt < 50) AND "SeqData".setStop1) OR (("SeqData".posCaseBelt < 75) AND NOT "SeqData".setStop1 AND "SeqData".setStop2 AND "SeqData".toLift1) OR (("SeqData".posCaseBelt < 100) AND NOT "SeqData".setStop2 AND NOT "SeqData".toLift1)) AND "SeqData".plantOn AND #statRisTrigClock THEN
       "SeqData".posCaseBelt := "SeqData".posCaseBelt + 1;
   END_IF;
END_REGION

REGION Network 3: case positon on lift 1
   IF ("SeqData".posLift1 < 60) AND "SeqData".plantOn AND true AND "SeqData".outLift1Up AND #statRisTrigClock AND NOT "SeqData".simActReactSupVis THEN
       "SeqData".posLift1 := "SeqData".posLift1 + 2;
   END_IF;
   IF ("SeqData".posLift1 > 0) AND "SeqData".plantOn AND true AND "SeqData".outLift1Down AND #statRisTrigClock AND NOT "SeqData".simActReactSupVis THEN
       "SeqData".posLift1 := "SeqData".posLift1 - 2;
   END_IF;
END_REGION

REGION Network 4: case positon on lift 2
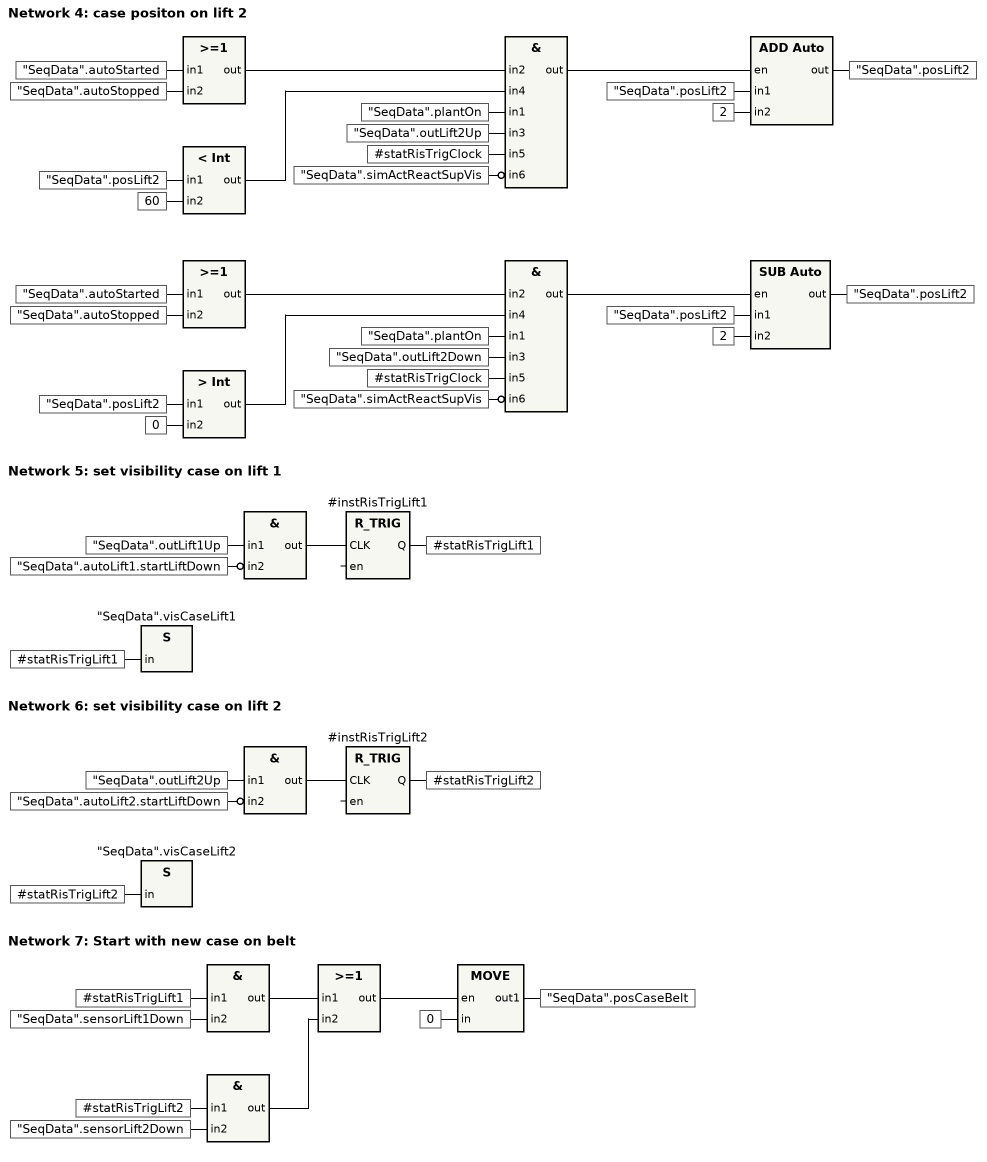
   IF ("SeqData".autoStarted OR "SeqData".autoStopped) AND ("SeqData".posLift2 < 60) AND "SeqData".plantOn AND "SeqData".outLift2Up AND #statRisTrigClock AND NOT "SeqData".simActReactSupVis THEN
       "SeqData".posLift2 := "SeqData".posLift2 + 2;
   END_IF;
   IF ("SeqData".autoStarted OR "SeqData".autoStopped) AND ("SeqData".posLift2 > 0) AND "SeqData".plantOn AND "SeqData".outLift2Down AND #statRisTrigClock AND NOT "SeqData".simActReactSupVis THEN
       "SeqData".posLift2 := "SeqData".posLift2 - 2;
   END_IF;
END_REGION

REGION Network 5: set visibility case on lift 1
   #instRisTrigLift1(CLK := "SeqData".outLift1Up AND NOT "SeqData".autoLift1.startLiftDown,   // R_TRIG
                     Q => #statRisTrigLift1);
   IF #statRisTrigLift1 THEN "SeqData".visCaseLift1 := TRUE; END_IF;
END_REGION

REGION Network 6: set visibility case on lift 2
   #instRisTrigLift2(CLK := "SeqData".outLift2Up AND NOT "SeqData".autoLift2.startLiftDown,   // R_TRIG
                     Q => #statRisTrigLift2);
   IF #statRisTrigLift2 THEN "SeqData".visCaseLift2 := TRUE; END_IF;
END_REGION

REGION Network 7: Start with new case on belt
   IF (#statRisTrigLift1 AND "SeqData".sensorLift1Down) OR (#statRisTrigLift2 AND "SeqData".sensorLift2Down) THEN
       "SeqData".posCaseBelt := 0;
   END_IF;
END_REGION

REGION Network 8: check, if new case
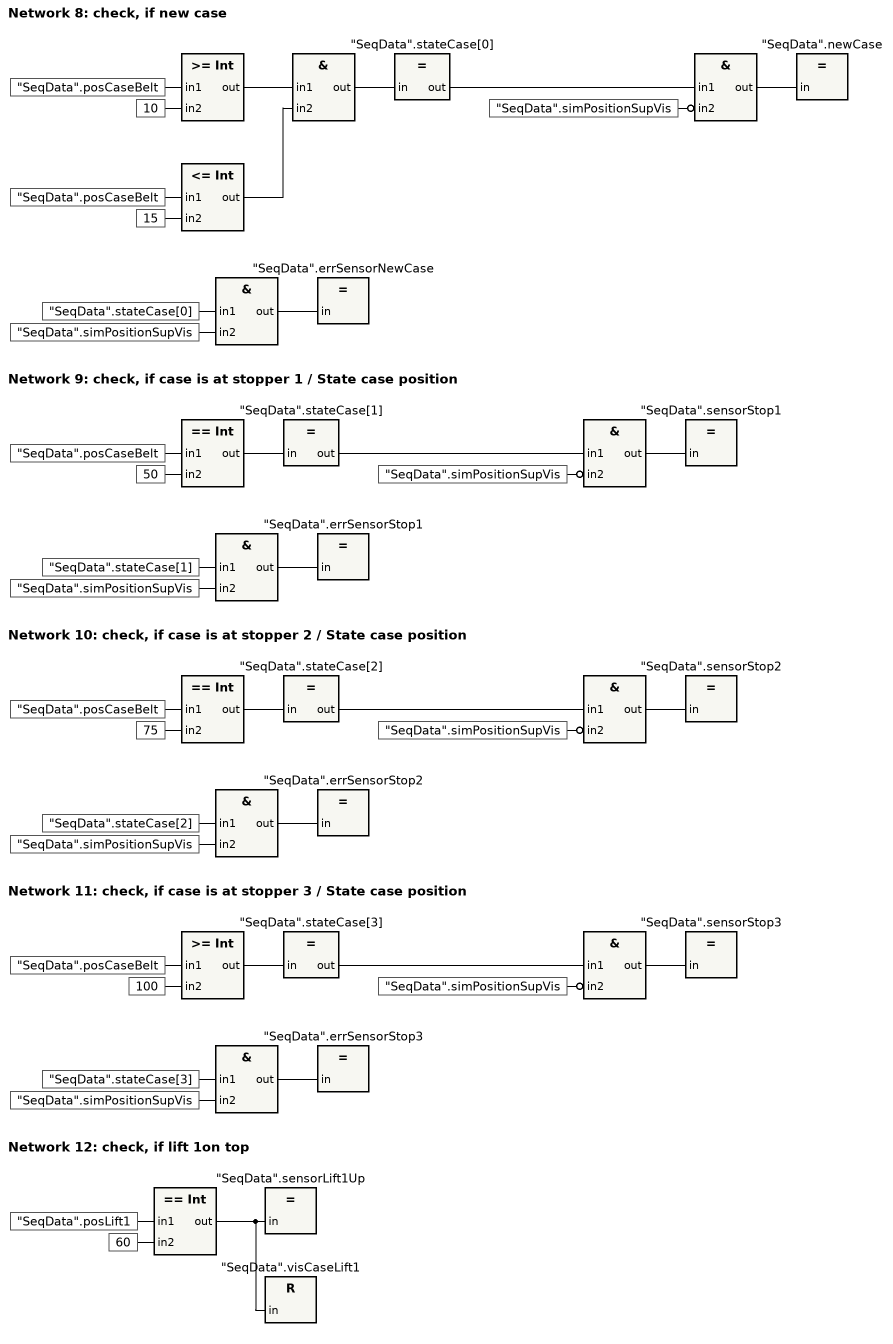
   "SeqData".stateCase[0] := ("SeqData".posCaseBelt >= 10) AND ("SeqData".posCaseBelt <= 15);
   "SeqData".newCase := ("SeqData".posCaseBelt >= 10) AND ("SeqData".posCaseBelt <= 15) AND NOT "SeqData".simPositionSupVis;
   "SeqData".errSensorNewCase := "SeqData".stateCase[0] AND "SeqData".simPositionSupVis;
END_REGION

REGION Network 9: check, if case is at stopper 1 / State case position
   "SeqData".stateCase[1] := "SeqData".posCaseBelt = 50;
   "SeqData".sensorStop1 := ("SeqData".posCaseBelt = 50) AND NOT "SeqData".simPositionSupVis;
   "SeqData".errSensorStop1 := "SeqData".stateCase[1] AND "SeqData".simPositionSupVis;
END_REGION

REGION Network 10: check, if case is at stopper 2 / State case position
   "SeqData".stateCase[2] := "SeqData".posCaseBelt = 75;
   "SeqData".sensorStop2 := ("SeqData".posCaseBelt = 75) AND NOT "SeqData".simPositionSupVis;
   "SeqData".errSensorStop2 := "SeqData".stateCase[2] AND "SeqData".simPositionSupVis;
END_REGION

REGION Network 11: check, if case is at stopper 3 / State case position
   "SeqData".stateCase[3] := "SeqData".posCaseBelt >= 100;
   "SeqData".sensorStop3 := ("SeqData".posCaseBelt >= 100) AND NOT "SeqData".simPositionSupVis;
   "SeqData".errSensorStop3 := "SeqData".stateCase[3] AND "SeqData".simPositionSupVis;
END_REGION

REGION Network 12: check, if lift 1on top
   "SeqData".sensorLift1Up := "SeqData".posLift1 = 60;
   IF "SeqData".sensorLift1Up THEN "SeqData".visCaseLift1 := FALSE; END_IF;
END_REGION

REGION Network 13: check, if lift 2 on top
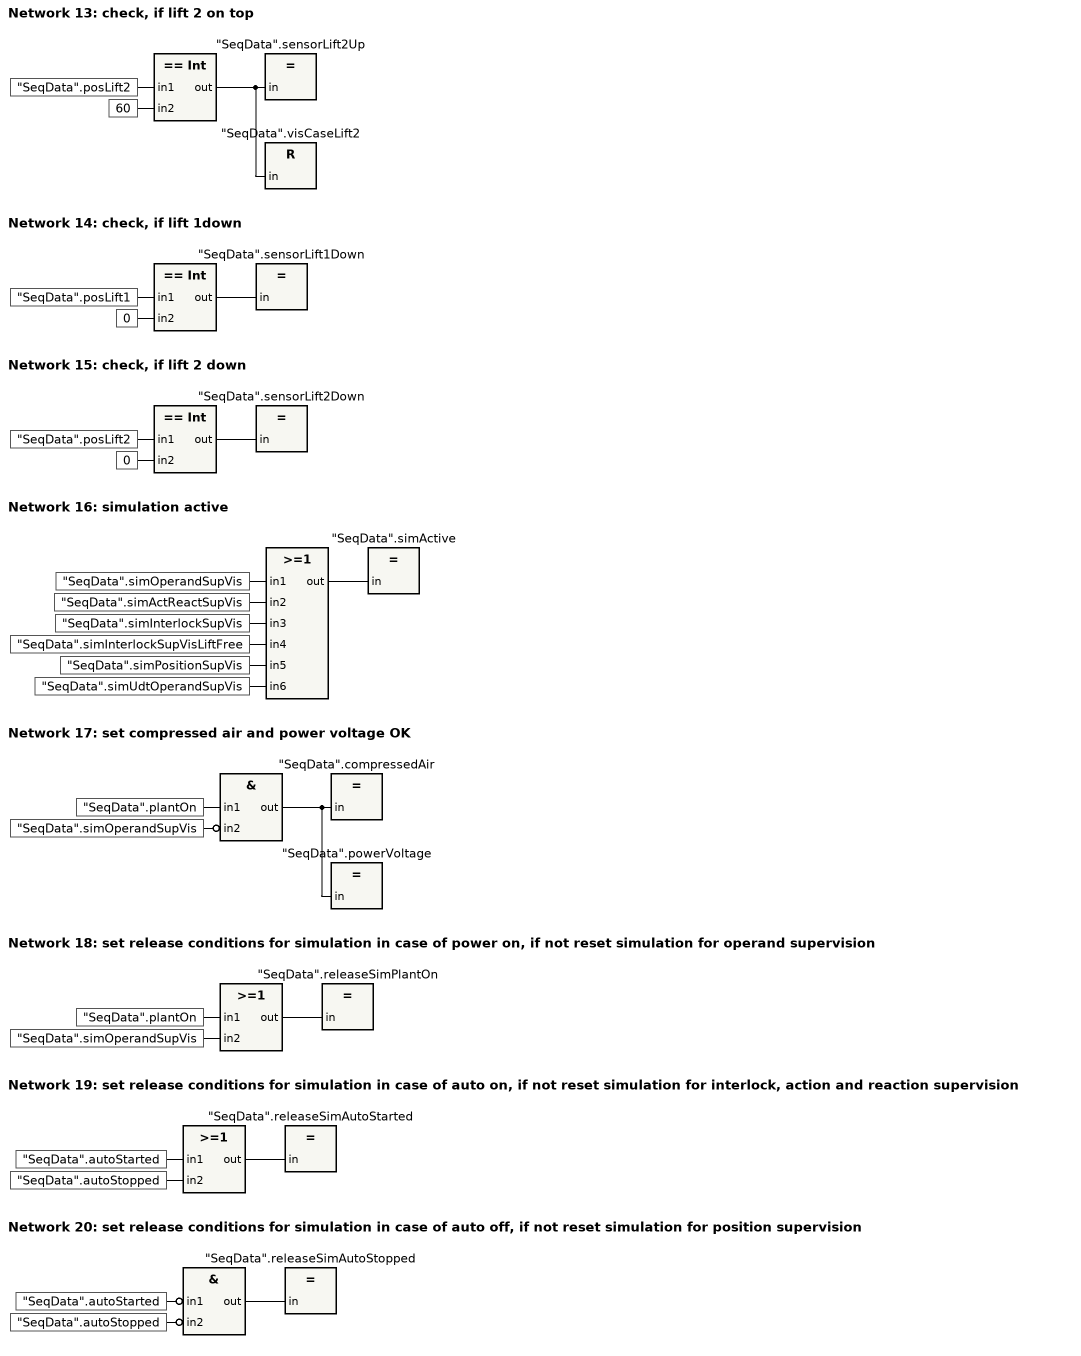
   "SeqData".sensorLift2Up := "SeqData".posLift2 = 60;
   IF "SeqData".sensorLift2Up THEN "SeqData".visCaseLift2 := FALSE; END_IF;
END_REGION

REGION Network 14: check, if lift 1down
   "SeqData".sensorLift1Down := "SeqData".posLift1 = 0;
END_REGION

REGION Network 15: check, if lift 2 down
   "SeqData".sensorLift2Down := "SeqData".posLift2 = 0;
END_REGION

REGION Network 16: simulation active
   "SeqData".simActive := "SeqData".simOperandSupVis OR "SeqData".simActReactSupVis OR "SeqData".simInterlockSupVis OR "SeqData".simInterlockSupVisLiftFree OR "SeqData".simPositionSupVis OR "SeqData".simUdtOperandSupVis;
END_REGION

REGION Network 17: set compressed air and power voltage OK
   "SeqData".compressedAir := "SeqData".plantOn AND NOT "SeqData".simOperandSupVis;
   "SeqData".powerVoltage := "SeqData".compressedAir;
END_REGION

REGION Network 18: set release conditions for simulation in case of power on, if not reset simulation for operand supervision
   "SeqData".releaseSimPlantOn := "SeqData".plantOn OR "SeqData".simOperandSupVis;
END_REGION

REGION Network 19: set release conditions for simulation in case of auto on, if not reset simulation for interlock, action and reaction supervision
   "SeqData".releaseSimAutoStarted := "SeqData".autoStarted OR "SeqData".autoStopped;
END_REGION

REGION Network 20: set release conditions for simulation in case of auto off, if not reset simulation for position supervision
   "SeqData".releaseSimAutoStopped := NOT "SeqData".autoStarted AND NOT "SeqData".autoStopped;
END_REGION

REGION Network 21: set door closed
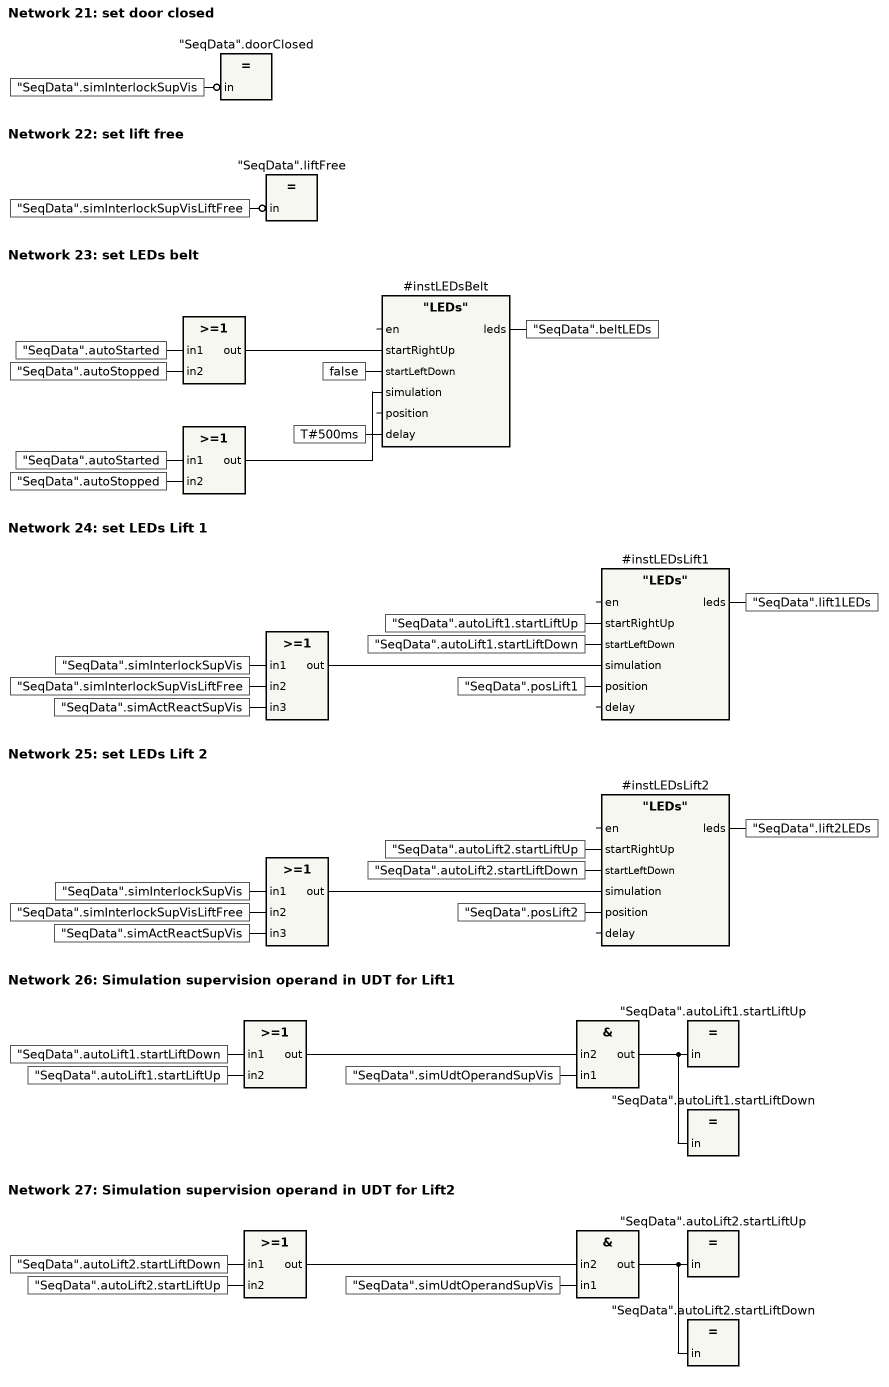
   "SeqData".doorClosed := NOT "SeqData".simInterlockSupVis;
END_REGION

REGION Network 22: set lift free
   "SeqData".liftFree := NOT "SeqData".simInterlockSupVisLiftFree;
END_REGION

REGION Network 23: set LEDs belt
   #instLEDsBelt(startRightUp := "SeqData".autoStarted OR "SeqData".autoStopped,   // "LEDs"
                 startLeftDown := false,
                 simulation := "SeqData".autoStarted OR "SeqData".autoStopped,
                 delay := T#500ms,
                 leds => "SeqData".beltLEDs);
END_REGION

REGION Network 24: set LEDs Lift 1
   #instLEDsLift1(startRightUp := "SeqData".autoLift1.startLiftUp,   // "LEDs"
                  startLeftDown := "SeqData".autoLift1.startLiftDown,
                  simulation := "SeqData".simInterlockSupVis OR "SeqData".simInterlockSupVisLiftFree OR "SeqData".simActReactSupVis,
                  position := "SeqData".posLift1,
                  leds => "SeqData".lift1LEDs);
END_REGION

REGION Network 25: set LEDs Lift 2
   #instLEDsLift2(startRightUp := "SeqData".autoLift2.startLiftUp,   // "LEDs"
                  startLeftDown := "SeqData".autoLift2.startLiftDown,
                  simulation := "SeqData".simInterlockSupVis OR "SeqData".simInterlockSupVisLiftFree OR "SeqData".simActReactSupVis,
                  position := "SeqData".posLift2,
                  leds => "SeqData".lift2LEDs);
END_REGION

REGION Network 26: Simulation supervision operand in UDT for Lift1
   "SeqData".autoLift1.startLiftUp := ("SeqData".autoLift1.startLiftDown OR "SeqData".autoLift1.startLiftUp) AND "SeqData".simUdtOperandSupVis;
   "SeqData".autoLift1.startLiftDown := "SeqData".autoLift1.startLiftUp;
END_REGION

REGION Network 27: Simulation supervision operand in UDT for Lift2
   "SeqData".autoLift2.startLiftUp := ("SeqData".autoLift2.startLiftDown OR "SeqData".autoLift2.startLiftUp) AND "SeqData".simUdtOperandSupVis;
   "SeqData".autoLift2.startLiftDown := "SeqData".autoLift2.startLiftUp;
END_REGION
END_FUNCTION_BLOCK

FUNCTION_BLOCK "Frequency"   // FB100, SCL
TITLE = Frequency
{ S7_Optimized_Access := 'TRUE' }
AUTHOR : Siemens
VERSION : 0.0.0.0
// Frequency (speed BeltLift)
// stored: IsIECCheckEnabled true, MemoryReserve 100, SetENOAutomatically true
   VAR_INPUT
      frequency { ExternalAccessible := 'False'; ExternalVisible := 'False'; ExternalWritable := 'False'} : Real := 10.0;   // Input in Hz
   END_VAR
   VAR_OUTPUT
      clock { ExternalAccessible := 'False'; ExternalVisible := 'False'; ExternalWritable := 'False'} : Bool;
      countdown { ExternalAccessible := 'False'; ExternalVisible := 'False'; ExternalWritable := 'False'} : Time;
      error { ExternalAccessible := 'False'; ExternalVisible := 'False'; ExternalWritable := 'False'} : Bool;
      status { ExternalAccessible := 'False'; ExternalVisible := 'False'; ExternalWritable := 'False'} : Word;
   END_VAR
   VAR
      instTofTimeOn { ExternalAccessible := 'False'; ExternalVisible := 'False'; ExternalWritable := 'False'; S7_SetPoint := 'True'} : TOF_TIME;
      instTofTimeOff { ExternalAccessible := 'False'; ExternalVisible := 'False'; ExternalWritable := 'False'; S7_SetPoint := 'True'} : TOF_TIME;
      statFrequencyMem { ExternalAccessible := 'False'; ExternalVisible := 'False'; ExternalWritable := 'False'} : Real;
      statTimeBase { ExternalAccessible := 'False'; ExternalVisible := 'False'; ExternalWritable := 'False'} : Time;
   END_VAR
   VAR CONSTANT
      MIN_FREQU : Real := 5.0;
      MAX_FREQU : Real := 10.0;
      FREQU_TO_LOW : Word := 16#8001;
      FREQU_TO_HIGH : Word := 16#8002;
   END_VAR
BEGIN
   //=============================================================================
   // Siemens AG
   // (c)Copyright 2015 All Rights Reserved
   //-----------------------------------------------------------------------------
   // Library:       LGF(Library General Functions)
   // Tested with:   CPU1212C DC/DC/DC FW:V4.1
   // Engineering:   TIA Portal V13 SP1 Upd 4
   // Restrictions:  -
   // Requirements:  PLC (S7-1200, S7-1500)
   // Functionality: Generates frequency signal
   //-----------------------------------------------------------------------------
   // Change log table:
   // Version  Date        Expert in charge                Changes applied
   // 01.00.00 21.07.2015  Siemens Industry Online Support First released version 
   //=============================================================================

   #error := FALSE;
   #status := 0;

   IF (#frequency <= 0.0)  // If input is <= 0.0 >> block is off // Wenn Eingang kleiner als 0.0 >> Baustein arbeitet nicht
   THEN
     #clock := FALSE;
     #countdown := t#0s;
   ELSE
     IF (#statFrequencyMem <> #frequency) // assign frequency one time   // Frequenz zuweisen
     THEN
       #statTimeBase := t#1000s / TRUNC(#frequency * 2000); // calculate time  //Zeit berechnen
       #statFrequencyMem := #frequency;
     END_IF;

     // TOF_off expired >> Start again // TOF_off abgelaufen starte von vorn
     #instTofTimeOn(IN := NOT #instTofTimeOff.Q,
                    PT := #statTimeBase);
     #countdown := #statTimeBase - #instTofTimeOn.ET;

     #instTofTimeOff(IN := #instTofTimeOn.Q,
                     PT := #statTimeBase);

     IF #countdown = t#0s THEN
       #countdown := #statTimeBase - #instTofTimeOff.ET;
     END_IF;

     #clock := #instTofTimeOn.Q; //assign ouptut // Frequenzausgang setzen   
   END_IF;

   //------------------------------------------------------------------------
   // Program for error message
   //------------------------------------------------------------------------
   IF (#frequency < #MIN_FREQU)
   THEN
     IF #status = 16#8002
     THEN
       #status := 0;
     ELSE
       #status := #FREQU_TO_LOW;
       #error := TRUE;
       RETURN;
     END_IF;
   END_IF;

   IF (#frequency > #MAX_FREQU)
   THEN
     IF #status = 16#8001
     THEN
       #status := 0;
     ELSE
       #status := #FREQU_TO_HIGH;
       #error := TRUE;
       RETURN;
     END_IF;
   END_IF;

   IF (#frequency = 10.0)
   THEN
     #status := 0;
     #error := 0;
     RETURN;
   END_IF;
END_FUNCTION_BLOCK

FUNCTION_BLOCK "LEDs"   // FB15, SCL
TITLE = LED
{ S7_Optimized_Access := 'TRUE' }
AUTHOR : Siemens
// LEDs BeltLift
// stored: IsIECCheckEnabled true, MemoryReserve 100, SetENOAutomatically true
   VAR_INPUT
      startRightUp { ExternalAccessible := 'False'; ExternalVisible := 'False'; ExternalWritable := 'False'} : Bool;
      startLeftDown { ExternalAccessible := 'False'; ExternalVisible := 'False'; ExternalWritable := 'False'} : Bool;
      simulation { ExternalAccessible := 'False'; ExternalVisible := 'False'; ExternalWritable := 'False'} : Bool;
      position { ExternalAccessible := 'False'; ExternalVisible := 'False'; ExternalWritable := 'False'} : Int;
      delay { ExternalAccessible := 'False'; ExternalVisible := 'False'; ExternalWritable := 'False'} : Time := T#400ms;
   END_VAR
   VAR_OUTPUT
      leds { ExternalAccessible := 'False'; ExternalVisible := 'False'; ExternalWritable := 'False'} : Word;
   END_VAR
   VAR
      instMovingLightLift { ExternalAccessible := 'False'; ExternalVisible := 'False'; ExternalWritable := 'False'; S7_SetPoint := 'True'} : "MovingLight";
      statDirLift { ExternalAccessible := 'False'; ExternalVisible := 'False'; ExternalWritable := 'False'} : Int;
   END_VAR
   VAR CONSTANT
      STOP : Int;
      LEFT_DOWN : Int := 10;
      RIGHT_UP : Int := 20;
   END_VAR
BEGIN
   IF #simulation
   THEN
     // set led direction
     IF #startRightUp
     THEN
       #statDirLift := #RIGHT_UP;
     ELSIF #startLeftDown
     THEN
       #statDirLift := #LEFT_DOWN;
     ELSE
       #statDirLift := #STOP;
     END_IF;

     // call "MovingLight"
     #instMovingLightLift(lightDirection := #statDirLift,
                          nBitsLight := 10,
                          delay := #delay,
                          wrd1 => #leds);

   ELSE

     CASE #position OF
       0:  
         #leds := 0;
       1..10:
         #leds := 1;
       11..20:
         #leds := 2;
       21..30:
         #leds := 4;
       31..40:
         #leds := 8;
       41..50:
         #leds := 16;
       51..60:
         #leds := 32;
       61..70:
         #leds := 64;
       71..80:
         #leds := 128;
       81..90:
         #leds := 256;
       91..100:
         #leds := 512;

       ELSE  // Statement section ELSE
         #leds := 0;
     END_CASE;

   END_IF;
END_FUNCTION_BLOCK

FUNCTION_BLOCK "MovingLight"   // FB16, SCL
TITLE = MovingLight
{ S7_Optimized_Access := 'TRUE' }
AUTHOR : Siemens
// Moving light BeltLift
// stored: IsIECCheckEnabled true, MemoryReserve 100, SetENOAutomatically true
   VAR_INPUT
      lightDirection { ExternalAccessible := 'False'; ExternalVisible := 'False'; ExternalWritable := 'False'} : Int;
      nBitsLight { ExternalAccessible := 'False'; ExternalVisible := 'False'; ExternalWritable := 'False'} : UInt;
      delay { ExternalAccessible := 'False'; ExternalVisible := 'False'; ExternalWritable := 'False'} : Time := T#200MS;   // Time delay for signal change
   END_VAR
   VAR_OUTPUT
      wrd1 { ExternalAccessible := 'False'; ExternalVisible := 'False'; ExternalWritable := 'False'} : Word;
   END_VAR
   VAR
      statDelayInt { ExternalAccessible := 'False'; ExternalVisible := 'False'; ExternalWritable := 'False'; S7_SetPoint := 'True'} : TOF_TIME;
      statGo { ExternalAccessible := 'False'; ExternalVisible := 'False'; ExternalWritable := 'False'} : Bool;
      statRun { ExternalAccessible := 'False'; ExternalVisible := 'False'; ExternalWritable := 'False'} : Time;
      statUp { ExternalAccessible := 'False'; ExternalVisible := 'False'; ExternalWritable := 'False'} : Word := 1;
      statMovingLight { ExternalAccessible := 'False'; ExternalVisible := 'False'; ExternalWritable := 'False'} : Word;
      statMaxMoveLightValue { ExternalAccessible := 'False'; ExternalVisible := 'False'; ExternalWritable := 'False'} : Word;
   END_VAR
   VAR CONSTANT
      STOP : Int;
      LEFT : Int := 10;
      RIGHT : Int := 20;
   END_VAR
BEGIN
   // function block for moving light with light direction left or right

   // calculate compare value dependent from number of LEDs used
   #statMaxMoveLightValue := 1;
   #statMaxMoveLightValue := SHL(IN := #statMaxMoveLightValue, N := (#nBitsLight - 1));

   // time delay
   #statDelayInt(IN := #statGo,
              PT := #delay,
              ET => #statRun);
   #statGo := NOT #statDelayInt.Q; // erneuter Start, wenn die Zeit abgelaufen ist


   CASE #lightDirection OF // Lauflichttypen auswählen
     #STOP:// no moving light
       #statUp := 0;

     #LEFT: // moving light left
       IF #statGo THEN
         #statMovingLight := SHR(IN := #statMovingLight, N := 1);

         IF (#statMovingLight = 0) THEN
           // set moving light to calculated value
           #statMovingLight := #statMaxMoveLightValue;
         END_IF;
         // change bytes
         // #up := SWAP(IN := #MovingLight); // SWAP only, if QW on output
         #statUp := #statMovingLight;
       END_IF;

     #RIGHT: // moving light right 
       IF #statGo THEN
         #statMovingLight := SHL(IN := #statMovingLight, N := 1);

         IF (#statMovingLight = 0) OR (#statMovingLight > #statMaxMoveLightValue) THEN
           // set first LED of moving light
           #statMovingLight := 1;
         END_IF;
         // change bytes
         // #up := SWAP(IN := #MovingLight); // SWAP only, if QW on output
         #statUp := #statMovingLight;
       END_IF;
     ELSE
       #statUp := 0;
   END_CASE;

   // output
   #wrd1 := #statUp;
END_FUNCTION_BLOCK

DATA_BLOCK "Block_1_DB"   // DB4
// stored: InstanceOfName Block_1, InstanceOfType FB
"Block_1"
   // VAR_INPUT
   //    V1 : Bool;
   // END_VAR
   // VAR
   //    Program_Alarm_1 { S7_SetPoint := 'True'} : Program_Alarm;
   // END_VAR
BEGIN
END_DATA_BLOCK

DATA_BLOCK "InstFrequency"   // DB2
TITLE = InstFrequncy
{ DB_Accessible_From_OPC_UA := 'FALSE' }
// IDB Frequency
// stored: AssignedProDiagFB LiftProDiagFB, DBAccessibleFromOPCUA false, InstanceOfName Frequency, InstanceOfType FB
"Frequency"
BEGIN
END_DATA_BLOCK

DATA_BLOCK "InstLiftSeq"   // DB12
TITLE = InstLiftSeq
{ DB_Accessible_From_OPC_UA := 'FALSE' }
// IDB LiftSeq
// stored: DBAccessibleFromOPCUA false, InstanceOfName LiftSeq, InstanceOfType FB
"LiftSeq"
BEGIN
END_DATA_BLOCK

DATA_BLOCK "InstMainFB"   // DB10
TITLE = InstMainFB
{ DB_Accessible_From_OPC_UA := 'FALSE' }
// IDB MainFB
// stored: AssignedProDiagFB LiftProDiagFB, DBAccessibleFromOPCUA false, InstanceOfName MainFB, InstanceOfType FB
"MainFB"
BEGIN
END_DATA_BLOCK
